# EPICS autosave request: iocs/xspress3IOC/iocBoot/iocXspress3/xsp3-4ch.req
file "xsp3.req", P=$(P)
file "xsp3_chan.req", P=$(P), CHAN=1
file "xsp3_chan.req", P=$(P), CHAN=2
file "xsp3_chan.req", P=$(P), CHAN=3
file "xsp3_chan.req", P=$(P), CHAN=4
